PROGRAM ControlHumidity
VAR
END_VAR

IF iHumidity < stepArray[iCurrentIndex].iHumidityValue-5 THEN
	O_bKanavapuhallinKosteutus := TRUE; // Do something to raise humidity
ELSIF iHumidity > stepArray[iCurrentIndex].iHumidityValue+5 THEN
	O_bKanavapuhallinKosteutus := FALSE; // Do something to decrease humidity
END_IF

END_PROGRAM

(* stored: Version 1.1.0.1, ProductVersion 3.1.4019.2
   POU ControlHumidity: Id {dcfda000-fb12-495a-a79b-d12a2ad9cac0}, SpecialFunc None *)
